SYSTEM nameless
  (* Version 1.0 *)
  APPLICATION namelessApp
    FBS
      E_PERMIT : E_PERMIT(PERMIT := None);
      E_CTU : E_CTU(PV := None, Q := None, CV := None);
      E_RESTART : E_RESTART;
    END_FBS
    EVENT_CONNECTIONS
      E_PERMIT.EO TO E_CTU.CU;
      E_RESTART.WARM TO E_PERMIT.EI;
    END_CONNECTIONS
    DATA_CONNECTIONS
      E_CTU.PV TO E_PERMIT.PERMIT;
    END_CONNECTIONS
  END_APPLICATION
END_SYSTEM
